// TwinCAT 3 PLC project Camera_lib
// Title: Cognex_Camera
// Company: Thomas More
// Author: Arno Joosen
// ProjectVersion: 0.1.2
// ProgramVersion: 3.1.4023.0
// libraries:
//   Buffer Lib, * (Thomas More)
//   Tc2_Standard, * (Beckhoff Automation GmbH)
//   Tc2_System, * (Beckhoff Automation GmbH)
//   Tc3_Module, * (Beckhoff Automation GmbH)
// project tree:
//   DUTs/CameraIO/ Acquisition_Control.TcDUT, Acquisition_Status_Register.TcDUT, Inspection_Control_Register.TcDUT, Inspection_Status_Register.TcDUT, SoftEvent.TcDUT, Soft_Event_Control.TcDUT
//   DUTs/ Camera_Error.TcDUT, Camera_Type.TcDUT, Cognex_Camera.TcDUT, Jobe_Name.TcDUT, Trigger_Error.TcDUT
//   DUTs/States/ Camera_State.TcDUT, Command_State.TcDUT, Job_State.TcDUT
//   / PlcTask.TcTTO
//   POUs/Buffer_Data/ Camera_Get_Bool.TcPOU, Camera_Get_Int.TcPOU, Camera_Get_Real.TcPOU, Camera_Get_String.TcPOU, Camera_Set_Bool.TcPOU, Camera_Set_Int.TcPOU, Camera_Set_Real.TcPOU
//   POUs/ Camera_ClearErrors.TcPOU, Camera_Init.TcPOU, Camera_Load_Job.TcPOU, Camera_Set_Input_Layout.TcPOU, Camera_Set_Ouput_Layout.TcPOU, Camera_Trigger.TcPOU, Camera_Update.TcPOU
//   SubFunctions/ Update_Command_State.TcPOU, Update_Jobe_State.TcPOU
//   Version/ Global_Version.TcGVL
// (motion and I/O tree: see PLC project rfid_lib)
// real-time tasks:
//   TASK PlcTask: cycle T#10ms, priority 20, ADS port 350
//   TASK PlcTask1: cycle T#10ms, priority 21, ADS port 351
//   TASK PlcTask2: cycle T#10ms, priority 22, ADS port 352
//   TASK PlcTask3: cycle T#10ms, priority 23, ADS port 353

CONFIGURATION Camera_lib
    RESOURCE PLC ON TwinCAT3
        TASK PlcTask(INTERVAL := T#10ms, PRIORITY := 21);
        PROGRAM MAIN WITH PlcTask : MAIN;
    END_RESOURCE
END_CONFIGURATION

// ---- DUTs/CameraIO/Acquisition_Control.TcDUT
TYPE Acquisition_Control :
STRUCT
	Acquistion_Trigger_Enable : BIT;
	Acquistion_Trigger : BIT;
	Clear_Exposure_Complete : BIT;
	Set_Offline : BIT;
END_STRUCT
END_TYPE

// ---- DUTs/CameraIO/Acquisition_Status_Register.TcDUT
TYPE Acquisition_Status_Register :
STRUCT
	Acquisition_Trigger_Ready : BIT;
	Acquistion_Trigger_Acknowledge : BIT;
	Exposure_Complete : BIT;
	Missed_Acquisition : BIT;
	Offline_Reason_0 : BIT;
	Offline_Reason_1 : BIT;
	Offline_Reason_2 : BIT;
	Online : BIT;
END_STRUCT
END_TYPE

// ---- DUTs/CameraIO/Inspection_Control_Register.TcDUT
TYPE Inspection_Control_Register :
STRUCT
	Enable_Results_Buffering : BIT;
	Acknowledge_Inspection_Results : BIT;
	Extended_User_Data_Set : BIT;
	Execute_Command : BIT;
	Clear_Error : BIT;
END_STRUCT
END_TYPE

// ---- DUTs/CameraIO/Inspection_Status_Register.TcDUT
TYPE Inspection_Status_Register :
STRUCT
	System_Busy : BIT;
	Inspection_Completed : BIT;
	Results_Buffer_Overrun : BIT;
	Results_Valid : BIT;
	Command_Executing : BIT;
	Command_Complete : BIT;
	Command_Failed : BIT;
	Exetended_User_Data_Set_Acknowledge : BIT;
	Pass : BIT;
	Test_Run_Ready : BIT;
	Error : BIT;
END_STRUCT
END_TYPE

// ---- DUTs/CameraIO/SoftEvent.TcDUT
TYPE SoftEvent :
STRUCT
	Soft_Event_0 : BIT;
	Soft_Event_1 : BIT;
	Soft_Event_2 : BIT;
	Soft_Event_3 : BIT;
	Soft_Event_4 : BIT;
	Soft_Event_5 : BIT;
	Soft_Event_6 : BIT;
	Soft_Event_7 : BIT;
END_STRUCT
END_TYPE

// ---- DUTs/CameraIO/Soft_Event_Control.TcDUT
TYPE Soft_Event_Control :
STRUCT
	Soft_Event_0 : BIT;
	Soft_Event_1 : BIT;
	Soft_Event_2 : BIT;
	Soft_Event_3 : BIT;
	Soft_Event_4 : BIT;
	Soft_Event_5 : BIT;
	Soft_Event_6 : BIT;
	Soft_Event_7 : BIT;
END_STRUCT
END_TYPE

// ---- DUTs/Camera_Error.TcDUT
{attribute 'qualified_only'}
{attribute 'strict'}
TYPE Camera_Error :
(
	None := 0,
	StateError := 1,
	Trigger_Set_While_disabeld := 2,
	Trigger_Set_While_Offline := 3,
	Already_Executing := 4,
	Job_Load_Requested_While_Online := 5,
	Job_Does_Not_Exist := 6,
	Time_Out := 7
) UINT;
END_TYPE

// ---- DUTs/Camera_Type.TcDUT
{attribute 'qualified_only'}
{attribute 'strict'}
TYPE Camera_Type :
(
	Cognex_7000 := 0,
	Cognex_5100 := 1
)UINT;
END_TYPE

// ---- DUTs/Cognex_Camera.TcDUT
TYPE Cognex_Camera :
STRUCT
	// IO
	AcquisitionControl AT %Q* : Acquisition_Control;
	AcquisitionStatusRegister AT %I* : Acquisition_Status_Register;
	AcquistionID AT %I* : UINT;
	InspectionControlRegister AT %Q* : Inspection_Control_Register;
	InspectionStatusRegister AT %I* : Inspection_Status_Register;
	ErrorCode AT %I* : UINT;
	CurrentJobID AT %I* : UINT;
	Command_B AT %Q* : UINT;
	Command AT%Q* : USINT;
	SoftEventStatus AT %I* : SoftEvent;
	SoftEventControl AT %Q* : SoftEvent;
	UserData AT %Q* : ARRAY[0..63] OF BYTE; // TODO grote bepalen on compile time
	InspectionID AT %I* : UINT;
	ResultCode AT %I* : UINT;
	InspectionResults AT %I* : ARRAY[0..63] OF BYTE; // TODO grote bepalen on compile time
	
	// local var
	Input_Buffer_Layout : Buffer_Layout;
	Ouput_Buffer_Layout : Buffer_Layout;
	CameraState : Camera_State := Camera_State.Idel;
	JobeState : Job_State;
	CommandState : Command_State;
	Error : Camera_Error := Camera_Error.None;
	CameraType : Camera_Type;
END_STRUCT
END_TYPE

// ---- DUTs/Jobe_Name.TcDUT
TYPE Jobe_Name :
UNION
	StrVal : STRING[63];
	ArayVal : ARRAY[0..63] OF BYTE;
END_UNION
END_TYPE

// ---- DUTs/States/Camera_State.TcDUT
{attribute 'qualified_only'}
{attribute 'strict'}
TYPE Camera_State :
(
	Idel := 0,
	Jope_Running := 1,
	Command_Running := 2,
	Error := 3,
	Clear_Error := 4
) UINT;
END_TYPE

// ---- DUTs/States/Command_State.TcDUT
{attribute 'qualified_only'}
{attribute 'strict'}
TYPE Command_State :
(
	Exekute := 0,
	Wate := 1,
	Complete := 2,
	Error := 3
) UINT;
END_TYPE

// ---- DUTs/States/Job_State.TcDUT
{attribute 'qualified_only'}
{attribute 'strict'}
TYPE Job_State :
(
	TriggerAck := 0,
	Wate := 1,
	Complte := 2,
	Error := 3
) UINT;
END_TYPE

// ---- DUTs/Trigger_Error.TcDUT
{attribute 'qualified_only'}
{attribute 'strict'}
TYPE Trigger_Error :
(
	None := 0,
	Camera_Busy := 1,
	Camera_Not_Trigger_Redy := 2
) UINT;
END_TYPE

// ---- Version/Global_Version.TcGVL
{attribute 'TcGenerated'}
{attribute 'no-analysis'}
{attribute 'linkalways'}
// This function has been automatically generated from the project information.
VAR_GLOBAL CONSTANT
	{attribute 'const_non_replaced'}
	stLibVersion_Cognex_Camera : ST_LibVersion := (iMajor := 0, iMinor := 1, iBuild := 2, iRevision := 0, nFlags := 0, sVersion := '0.1.2');
END_VAR

// ---- POUs/Buffer_Data/Camera_Get_Bool.TcPOU
FUNCTION Camera_Get_Bool : Buffer_Error
VAR_INPUT
	Camera : REFERENCE TO Cognex_Camera;
	Num : USINT;
END_VAR

VAR_IN_OUT
	Out : BOOL;
END_VAR

Camera_Get_Bool := Get_Bool_From_Buffer(Num:= Num, 
										Layout:= Camera.Ouput_Buffer_Layout, 
										Buffer:= Camera.User_Data.Data, 
										Out:= Out);

END_FUNCTION

// ---- POUs/Buffer_Data/Camera_Get_Int.TcPOU
FUNCTION Camera_Get_Int : Buffer_Error
VAR_INPUT
	Camera : REFERENCE TO Cognex_Camera;
	Num : USINT;
END_VAR

VAR_IN_OUT
	Out : INT;
END_VAR

Camera_Get_Int := Get_Int_From_Buffer(	Num:= Num, 
										Layout:= Camera.Input_Buffer_Layout, 
										Buffer:= Camera.User_Data.Data, 
										Out:= Out);

END_FUNCTION

// ---- POUs/Buffer_Data/Camera_Get_Real.TcPOU
FUNCTION Camera_Get_Real : Buffer_Error
VAR_INPUT
	Camera : REFERENCE TO Cognex_Camera;
	Num : USINT;
END_VAR

VAR_IN_OUT
	Out : REAL;
END_VAR

Camera_Get_Real := Get_Real_From_Buffer(Num:= Num, 
										Layout:= Camera.Input_Buffer_Layout, 
										Buffer:= Camera.User_Data.Data, 
										Out:= Out);

END_FUNCTION

// ---- POUs/Buffer_Data/Camera_Get_String.TcPOU
FUNCTION Camera_Get_String : Buffer_Error
VAR_INPUT
	Camera : REFERENCE TO Cognex_Camera;
	Num : USINT;
END_VAR
VAR_IN_OUT
	Out : STRING[8];
END_VAR

Camera_Get_String := Get_String_From_Buffer(Num:= Num, 
											Layout:= Camera.Input_Buffer_Layout, 
											Buffer:= Camera.User_Data.Data, 
											Out:= Out)

END_FUNCTION

// ---- POUs/Buffer_Data/Camera_Set_Bool.TcPOU
FUNCTION Camera_Set_Bool : Buffer_Error
VAR_INPUT
	Num : USINT;
	In : BOOL;
END_VAR

VAR_IN_OUT
	Camera : Cognex_Camera;
END_VAR

Camera_Set_Bool := Set_Bool_Fom_Buffer(	In:= In, 
										Num:= Num, 
										Layout:= Camera.Ouput_Buffer_Layout, 
										Buffer:= Camera.User_Data.UserData)

END_FUNCTION

// ---- POUs/Buffer_Data/Camera_Set_Int.TcPOU
FUNCTION Camera_Set_Int : Buffer_Error
VAR_INPUT
	Num : USINT;
	In : INT;
END_VAR

VAR_IN_OUT
	Camera : Cognex_Camera;
END_VAR

Camera_Set_Int := Set_Int_From_Buffer(	In:= In, 
										Num:= Num, 
										Layout:= Camera.Ouput_Buffer_Layout, 
										Buffer:= Camera.User_Data.UserData);

END_FUNCTION

// ---- POUs/Buffer_Data/Camera_Set_Real.TcPOU
FUNCTION Camera_Set_Real : Buffer_Error
VAR_INPUT
	Num : USINT;
	In : REAL;
END_VAR

VAR_IN_OUT
	Camera : Cognex_Camera;
END_VAR

Camera_Set_Real := Set_Real_From_Buffer(In:= In, 
										Num:= Num, 
										Layout:= Camera.Ouput_Buffer_Layout, 
										Buffer:= Camera.User_Data.UserData);

END_FUNCTION

// ---- POUs/Camera_ClearErrors.TcPOU
FUNCTION Camera_ClearErrors : BOOL
VAR_IN_OUT
	Camera : Cognex_Camera;
END_VAR

IF Camera.CameraState := Camera_State.Error THEN
	Camera.InspectionControlRegister.Clear_Error := TRUE;
	Camera.CameraState := Camera_State.Clear_Error;
END_IF

END_FUNCTION

// ---- POUs/Camera_Init.TcPOU
FUNCTION Camera_Init : BOOL
VAR_INPUT
	CameraType : Camera_Type;
END_VAR
VAR_IN_OUT
	Camera : Cognex_Camera;
END_VAR

Camera.AcquisitionControl.Acquistion_Trigger_Enable := TRUE;
Camera.CameraState := Camera_State.Idel;
Camera.CameraType := CameraType;

END_FUNCTION

// ---- POUs/Camera_Load_Job.TcPOU
FUNCTION Camera_Load_Job : BOOL
VAR_INPUT
	JobeName : STRING[63]; // 0..63 met 0 terminator
END_VAR
VAR_IN_OUT
	Camera : Cognex_Camera;
END_VAR
VAR
	i : UINT;
	UJobeName : Jobe_Name;
	End : BOOL := FALSE;
END_VAR

IF Camera.CameraState = Camera_State.Idel AND Camera.CameraType = Camera_Type.Cognex_7000 THEN
	// set camera in offline mode
	Camera.AcquisitionControl.Set_Offline := TRUE;
	// set command to load job by name
	Camera.Command_B := 16#4000;
	// load name in input user buffer
	UJobeName.StrVal := JobeName;
	FOR i:=0 TO 63 BY 1 DO
		IF UJobeName.StrVal[i] = 0 AND End THEN
			Camera.UserData[i] := 16#0; // set End
			End := TRUE;
		ELSE
			Camera.UserData[i] := UJobeName.StrVal[i];
		END_IF
	END_FOR
	// set execute
	Camera.CameraState := Camera_State.Command_Running;
	Camera.CommandState := Command_State.Set;
	Camera_Load_Job := TRUE;
ELSE
	Camera_Load_Job := FALSE;
END_IF

END_FUNCTION

// ---- POUs/Camera_Set_Input_Layout.TcPOU
FUNCTION Camera_Set_Input_Layout : UINT
VAR_INPUT
	Layout : Buffer_Layout;
END_VAR
VAR_IN_OUT
	Camera : Cognex_Camera;
END_VAR

Camera.Input_Buffer_Layout := Layout;

END_FUNCTION

// ---- POUs/Camera_Set_Ouput_Layout.TcPOU
FUNCTION Camera_Set_Ouput_Layout : UINT
VAR_INPUT
	Layout : Buffer_Layout;
END_VAR
VAR_IN_OUT
	Camera : Cognex_Camera;
END_VAR

Camera.Ouput_Buffer_Layout := Layout;

END_FUNCTION

// ---- POUs/Camera_Trigger.TcPOU
FUNCTION Camera_Trigger : Trigger_Error
VAR_IN_OUT
	Camera : Cognex_Camera;
END_VAR

IF Camera.CameraState = Camera_State.Idel THEN
	IF Camera.AcquisitionStatusRegister.Acquisition_Trigger_Ready THEN
		Camera.AcquisitionControl.Clear_Exposure_Complete := TRUE;
		Camera.AcquisitionControl.Acquistion_Trigger := TRUE;
		Camera.CameraState := Camera_State.Jope_Running;
		Camera.JobeState := Job_State.TriggerAck;
		Camera_Trigger := Trigger_Error.None;
	ELSE
		Camera_Trigger := Trigger_Error.Camera_Not_Trigger_Redy;
	END_IF
ELSE
	Camera_Trigger := Trigger_Error.Camera_Busy;
	RETURN;
END_IF

END_FUNCTION

// ---- POUs/Camera_Update.TcPOU
FUNCTION Camera_Update : Camera_Error
VAR_IN_OUT
	Camera : Cognex_Camera;
END_VAR

IF Camera.CameraState = Camera_State.Idel THEN
	RETURN;
ELSIF Camera.CameraState = Camera_State.Jope_Running THEN
	Update_Jobe_State(Camera);
ELSIF Camera.CameraState = Camera_State.Command_Running THEN
	Update_Command_State(Camera);
ELSIF Camera.CameraState = Camera_State.Clear_Error THEN
	Camera.InspectionControlRegister.Clear_Error := FALSE;
	Camera.CameraState := Camera_State.Idel;
ELSE
	Camera_Update := Camera.Error;
END_IF

END_FUNCTION

// ---- SubFunctions/Update_Jobe_State.TcPOU
FUNCTION Update_Jobe_State : BOOL
VAR_INPUT
	Camera : REFERENCE TO Cognex_Camera;
END_VAR
VAR
END_VAR

IF NOT Camera.CameraState = Camera_State.Jope_Running THEN
	RETURN;
END_IF

IF Camera.JobeState = Job_State.TriggerAck THEN
	IF Camera.AcquisitionStatusRegister.Acquistion_Trigger_Acknowledge THEN
		Camera.JobeState := Job_State.Wate;
		Camera.AcquisitionControl.Clear_Exposure_Complete := FALSE;
		Camera.AcquisitionControl.Acquistion_Trigger := FALSE;
		RETURN;
	ELSE
		RETURN;
	END_IF
ELSIF Camera.JobeState = Job_State.Wate THEN
	IF Camera.InspectionStatusRegister.Inspection_Completed AND (NOT Camera.InspectionStatusRegister.System_Busy) THEN
		Camera.JobeState := Job_State.Complte;
	END_IF
	
ELSIF Camera.InspectionStatusRegister.Error THEN
	Camera.JobeState := Job_State.Error;
	Camera.CameraState := Camera_State.Error;
	CASE Camera.ErrorCode OF
		16#0100: // Trigger set while disabeld
			Camera.Error := Camera_Error.Trigger_Set_While_disabeld;
		16#0101: // trigger set while offline
			Camera.Error := Camera_Error.Trigger_Set_While_Offline;
		16#0400: // already executing error
			Camera.Error := Camera_Error.Already_Executing;
		16#0401: // job load requeted while online
			Camera.Error := Camera_Error.Job_Load_Requested_While_Online;
		16#0402: // job load requested does not exist on the camera
			Camera.Error := Camera_Error.Job_Does_Not_Exist;
	END_CASE
ELSIF Camera.JobeState = Job_State.Error OR Camera.JobeState = Job_State.Complte THEN
	RETURN;
ELSE
	Camera.JobeState := Job_State.Error;
	Camera.Error := Camera_Error.StateError;
	RETURN;
END_IF

END_FUNCTION

// ---- SubFunctions/Update_Command_State.TcPOU
FUNCTION Update_Command_State : BOOL
VAR_INPUT
	Camera : REFERENCE TO Cognex_Camera;
END_VAR
VAR
END_VAR

IF Camera.CommandState = Command_State.Set THEN
	IF NOT Camera.AcquisitionStatusRegister.Online THEN
		Camera.InspectionControlRegister.Execute_Command := TRUE;
		Camera.CommandState := Command_State.Exekute;
	ELSE
		RETURN;
	END_IF;
ELSIF Camera.CommandState = Command_State.Exekute THEN
	Camera.InspectionControlRegister.Execute_Command := FALSE;
	Camera.CommandState := Command_State.Wate;
ELSIF Camera.CommandState = Command_State.Wate THEN
	IF Camera.InspectionStatusRegister.Command_Complete THEN
		Camera.CommandState := Command_State.Complete;
		Camera.InspectionControlRegister.Execute_Command := FALSE;
	ELSIF Camera.InspectionStatusRegister.Command_Failed THEN
		Camera.CommandState := Command_State.Error;
		Camera.CameraState := Camera_State.Error;
		Camera.InspectionControlRegister.Execute_Command := FALSE;
		CASE Camera.ErrorCode OF
			16#0100: // Trigger set while disabeld
				Camera.Error := Camera_Error.Trigger_Set_While_disabeld;
			16#0101: // trigger set while offline
				Camera.Error := Camera_Error.Trigger_Set_While_Offline;
			16#0400: // already executing error
				Camera.Error := Camera_Error.Already_Executing;
			16#0401: // job load requeted while online
				Camera.Error := Camera_Error.Job_Load_Requested_While_Online;
			16#0402: // job load requested does not exist on the camera
				Camera.Error := Camera_Error.Job_Does_Not_Exist;
		END_CASE
		RETURN;
	END_IF
ELSIF Camera.CommandState = Command_State.Error THEN
	Camera.CommandState := Command_State.Error;
	Camera.CameraState := Camera_State.Error;
	CASE Camera.ErrorCode OF
		16#0100: // Trigger set while disabeld
			Camera.Error := Camera_Error.Trigger_Set_While_disabeld;
		16#0101: // trigger set while offline
			Camera.Error := Camera_Error.Trigger_Set_While_Offline;
		16#0400: // already executing error
			Camera.Error := Camera_Error.Already_Executing;
		16#0401: // job load requeted while online
			Camera.Error := Camera_Error.Job_Load_Requested_While_Online;
		16#0402: // job load requested does not exist on the camera
			Camera.Error := Camera_Error.Job_Does_Not_Exist;
	END_CASE
	RETURN;
ELSE
	Camera.CommandState := Command_State.Error;
	Camera.Error := Camera_Error.StateError;
	RETURN;
END_IF

END_FUNCTION
